FUNCTION_BLOCK RingTokenMemberHead (* Basic Function Block Type *)
  (* Standard: 61499-2 *)
  (* Version 0.2, 2003-12-04, JHC, Rockwell Automation, Renamed for better indexing. *)
  (* Version 0.1, 2002-11-05, JHC, Rockwell Automation, Corrected missing ST element in Algorithm REQ. *)
  (* Version 0.0, 2000-05-30, JHC, Rockwell Automation *)
  (* Compiler header: package fb.rt.cs725; *)
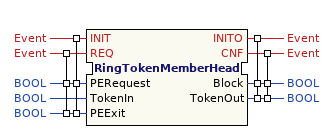
  EVENT_INPUT
    INIT WITH PERequest, PEExit; (* Initialization Request *)
    REQ WITH PERequest, PEExit; (* Normal Execution Request *)
  END_EVENT
  EVENT_OUTPUT
    INITO WITH Block, TokenOut; (* Initialization Confirm *)
    CNF WITH Block, TokenOut; (* Execution Confirmation *)
  END_EVENT
  VAR_INPUT
    PERequest : BOOL; (* Input event qualifier *)
    TokenIn : BOOL;
    PEExit : BOOL;
  END_VAR
  VAR_OUTPUT
    Block : BOOL; (* Output event qualifier *)
    TokenOut : BOOL;
  END_VAR
  VAR
    lastTokenIn : BOOL := 0;
    lastPEExit : BOOL := 0;
  END_VAR
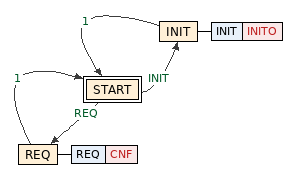
  EC_STATES
    START; (* Initial State *)
    INIT : INIT -> INITO; (* Initialization *)
    REQ : REQ -> CNF; (* Normal execution *)
  END_STATES
  EC_TRANSITIONS
    START TO INIT := INIT;
    INIT TO START := 1;
    START TO REQ := REQ;
    REQ TO START := 1;
  END_TRANSITIONS
  ALGORITHM INIT IN Java: (* Initialization algorithm *)
Block.value=false;
TokenOut.value=true;
System.out.println("init head, grant false, token true");
  END_ALGORITHM
  ALGORITHM REQ IN Java: (* Normally executed algorithm *)
boolean TokenChanged;
if (TokenIn.value != lastTokenIn.value) {
 TokenChanged = true;
} else {
 TokenChanged = false;
}

if (TokenChanged) {
 if (TokenIn.value) {
  if (!PERequest.value) {
   if (PEExit.value != lastPEExit.value) {
    if (PEExit.value) {
     Block.value = true;
     TokenOut.value = true;
     System.out.println("Conv 1 exiting critical section");
    }
    else {
        Block.value = false;
        TokenOut.value = false;
        System.out.println("Conv 1 entering/in critical section");
    }
   } else {
    Block.value = false;
    TokenOut.value = false;
    System.out.println("Conv 1 entering/in critical section");
   }
  } else {
   Block.value = false;
   TokenOut.value = true;
   System.out.println("2 Conv 1");
  }
 } else {
  TokenOut.value = false;
  Block.value = true;
  System.out.println("TokenChanged: " + this + " " + TokenIn.value);
 }
}

System.out.println("Current PEExit Value new/old conv 1: " + PEExit.value + "/" + lastPEExit.value)
  END_ALGORITHM
END_FUNCTION_BLOCK
